Fanuc KAREL source: ko00038.KL

PROGRAM KO00038
%STACKSIZE=65535
%PRIORITY=65535
%NOLOCKGROUP
VAR
P1 : POSITION
P2 : XYZWPR
F : BOOLEAN
OUT : XYZWPR
BEGIN
F=TRUE
-- UNSAFE_SOURCE_IR line 11: OUT = MIRROR(convert_position_to_xyzwprext(P1), convert_xyzwpr_to_position(P2), F)
END KO00038
